(* IEC 61131-3 sources: RL_MAR/experiments/comparison/autoplc/results/deepseek-ai-DeepSeek-V3.2_20260508_111905/med_56, 1 file *)

(* ---- med_56_1.st ---- *)
FUNCTION_BLOCK FB_SimpleRepeat
VAR_INPUT
    INPUT_VAR1 : INT := 2;
    INPUT_COUNTER : INT := 4;
END_VAR

VAR_OUTPUT
    OUTPUT_VAR1 : INT;
END_VAR

VAR
    COUNTER : INT;
END_VAR

    // Initialize counter and output
    COUNTER := INPUT_COUNTER;
    OUTPUT_VAR1 := INPUT_VAR1;

    // REPEAT loop implementation
    REPEAT
        OUTPUT_VAR1 := OUTPUT_VAR1 * 2;
        COUNTER := COUNTER - 1;
    UNTIL COUNTER = 0
    END_REPEAT;

END_FUNCTION_BLOCK
